# EPICS autosave request: apps/cRioApp/Db/gas_cRIO_SVT.req
#
# gas_cRIO_SVT.req - autosave alarm settings
#
$(P)$(R)N2SupFlow.LOLO
$(P)$(R)N2SupFlow.LOW
$(P)$(R)N2SupFlow.HIGH
$(P)$(R)N2SupFlow.HIHI
$(P)$(R)N2SupFlow.LLSV
$(P)$(R)N2SupFlow.LSV
$(P)$(R)N2SupFlow.HSV
$(P)$(R)N2SupFlow.HHSV
#
